PROGRAM MAIN
VAR
    suite : FB_SchmittTriggerTests;
END_VAR

suite();
TcUnit.RUN();

END_PROGRAM

(* stored: Version 1.1.0.1
   POU MAIN: Id {f427b895-601e-4ec8-b38b-44fdcf4e39a4}, SpecialFunc None *)
